FUNCTION_BLOCK FB_HeatingLoop
VAR_INPUT
	rPID_Core				: REAL;
	rPID_Surface			: REAL;
	ab_Sim_HE_Fault			: ARRAY [1..12] OF BOOL;
END_VAR
VAR_OUTPUT
	iOUT_Temperature_Core		: INT;
	iOUT_Temperature_Surface	: INT;
	abOUT_HE_Fault				: ARRAY [1..12] OF BOOL;
END_VAR
VAR
	FB_Sim_Core_1			: FB_PID_Simulation;
	FB_Sim_Core_2			: FB_PID_Simulation;
	FB_Sim_Surface_1		: FB_PID_Simulation;
	FB_Sim_Surface_2		: FB_PID_Simulation;
	
	rTemperature_Core		: REAL;
	rTemperatrue_Surface	: REAL;
	
// Temp Variables
	rTempC				: REAL;
	rTempC_2			: REAL;
	rPID_Core_Temp		: REAL;
	rTempS				: REAL;
	rTempS_2			: REAL;

END_VAR
VAR // added by the converter: edge detectors and wires of the graphical bodies
    _w1 : BOOL;
END_VAR

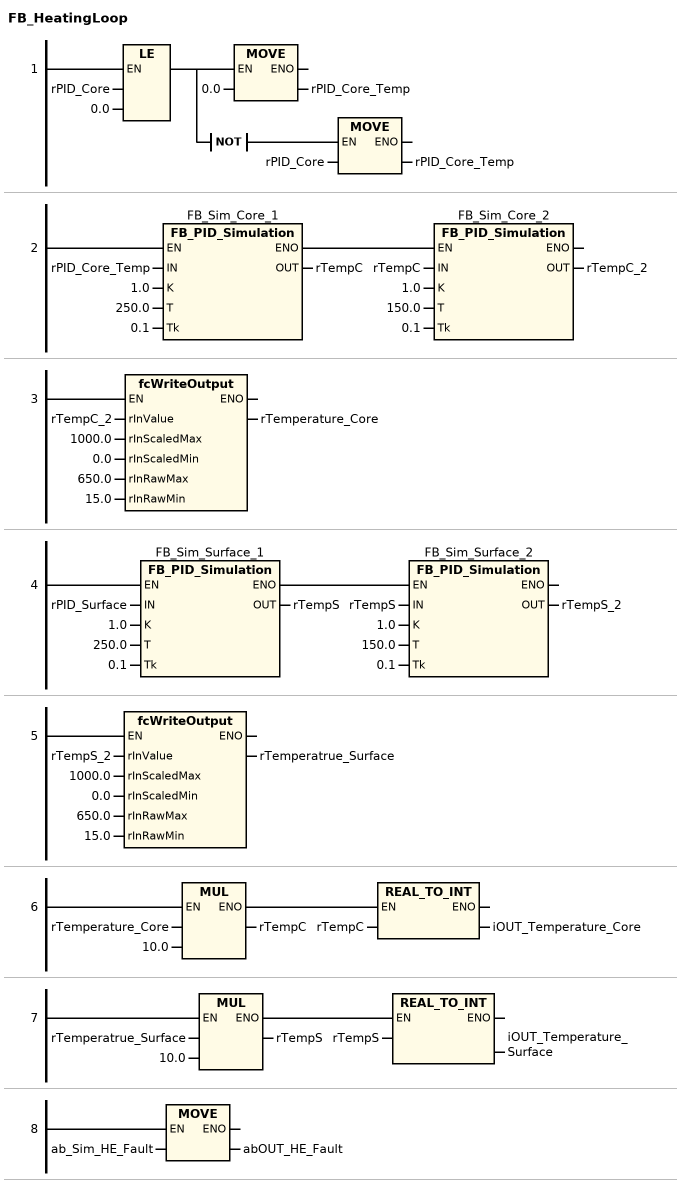
// NETWORK 1
_w1 := rPID_Core <= 0.0;
IF _w1 THEN rPID_Core_Temp := 0.0; END_IF
IF NOT _w1 THEN rPID_Core_Temp := rPID_Core; END_IF

// NETWORK 2
FB_Sim_Core_1(IN := rPID_Core_Temp, K := 1.0, T := 250.0, Tk := 0.1, OUT => rTempC); // FB_PID_Simulation
FB_Sim_Core_2(IN := rTempC, K := 1.0, T := 150.0, Tk := 0.1, OUT => rTempC_2); // FB_PID_Simulation

// NETWORK 3
rTemperature_Core := fcWriteOutput(rInValue := rTempC_2, rInScaledMax := 1000.0, rInScaledMin := 0.0, rInRawMax := 650.0, rInRawMin := 15.0);

// NETWORK 4
FB_Sim_Surface_1(IN := rPID_Surface, K := 1.0, T := 250.0, Tk := 0.1, OUT => rTempS); // FB_PID_Simulation
FB_Sim_Surface_2(IN := rTempS, K := 1.0, T := 150.0, Tk := 0.1, OUT => rTempS_2); // FB_PID_Simulation

// NETWORK 5
rTemperatrue_Surface := fcWriteOutput(rInValue := rTempS_2, rInScaledMax := 1000.0, rInScaledMin := 0.0, rInRawMax := 650.0, rInRawMin := 15.0);

// NETWORK 6
rTempC := rTemperature_Core * 10.0;
iOUT_Temperature_Core := REAL_TO_INT(rTempC);

// NETWORK 7
rTempS := rTemperatrue_Surface * 10.0;
iOUT_Temperature_Surface := REAL_TO_INT(rTempS);

// NETWORK 8
abOUT_HE_Fault := ab_Sim_HE_Fault;

END_FUNCTION_BLOCK

(* stored: Version 1.1.0.1, ProductVersion 3.1.4024.12
   POU FB_HeatingLoop: Id {309fcbc1-1026-4dda-bc18-07e4f1dd634b}, SpecialFunc None *)
